LIN {X 0,Y 100.79,Z 485.874,A -85,B 0,C 180,E1 -28454.124,E2 -28454.124} C_VEL
LIN {X 0,Y 100.608,Z 489.017,A -85,B 0,C 180,E1 -28458.321,E2 -28458.321} C_VEL
LIN {X 0,Y 99.957,Z 495.022,A -85,B 0,C 180,E1 -28464.952,E2 -28464.952} C_VEL
LIN {X 0,Y 99.623,Z 497.358,A -85,B 0,C 180,E1 -28467.293,E2 -28467.293} C_VEL
LIN {X 0,Y 98.959,Z 499.354,A -85,B 0,C 180,E1 -28468.917,E2 -28468.917} C_VEL
LIN {X 0,Y 94.552,Z 506.247,A -85,B 0,C 180,E1 -28473.257,E2 -28473.257} C_VEL
LIN {X 0,Y 91.523,Z 510.415,A -85,B 0,C 180,E1 -28476.263,E2 -28476.263} C_VEL
LIN {X 0,Y 84.205,Z 517.353,A -85,B 0,C 180,E1 -28481.307,E2 -28481.307} C_VEL
LIN {X 0,Y 77.66,Z 522.926,A -85,B 0,C 180,E1 -28487.255,E2 -28487.255} C_VEL
LIN {X 0,Y 72.027,Z 527.307,A -85,B 0,C 180,E1 -28494.164,E2 -28494.164} C_VEL
LIN {X 0,Y 68.844,Z 529.631,A -85,B 0,C 180,E1 -28499.307,E2 -28499.307} C_VEL
LIN {X 0,Y 66.338,Z 531.525,A -85,B 0,C 180,E1 -28504.927,E2 -28504.927} C_VEL
LIN {X 0,Y 63.396,Z 533.992,A -85,B 0,C 180,E1 -28517.189,E2 -28517.189} C_VEL
LIN {X 0,Y 62.912,Z 534.633,A -85,B 0,C 180,E1 -28523.585,E2 -28523.585} C_VEL
LIN {X 0,Y 63.099,Z 534.874,A -85,B 0,C 180,E1 -28529.999,E2 -28529.999} C_VEL
LIN {X 0,Y 62.911,Z 534.616,A -85,B 0,C 180,E1 -28536.414,E2 -28536.414} C_VEL
LIN {X 0,Y 63.389,Z 533.964,A -85,B 0,C 180,E1 -28542.811,E2 -28542.811} C_VEL
LIN {X 0,Y 66.335,Z 531.47,A -85,B 0,C 180,E1 -28555.073,E2 -28555.073} C_VEL
LIN {X 0,Y 70.389,Z 528.468,A -85,B 0,C 180,E1 -28563.308,E2 -28563.308} C_VEL
LIN {X 0,Y 75.675,Z 524.426,A -85,B 0,C 180,E1 -28570.549,E2 -28570.549} C_VEL
LIN {X 0,Y 82.981,Z 518.283,A -85,B 0,C 180,E1 -28577.722,E2 -28577.722} C_VEL
LIN {X 0,Y 90.316,Z 511.485,A -85,B 0,C 180,E1 -28582.903,E2 -28582.903} C_VEL
LIN {X 0,Y 93.523,Z 507.46,A -85,B 0,C 180,E1 -28585.753,E2 -28585.753} C_VEL
LIN {X 0,Y 98.232,Z 500.238,A -85,B 0,C 180,E1 -28590.434,E2 -28590.434} C_VEL
LIN {X 0,Y 98.86,Z 499.173,A -85,B 0,C 180,E1 -28591.096,E2 -28591.096} C_VEL
LIN {X 0,Y 99.501,Z 497.198,A -85,B 0,C 180,E1 -28592.701,E2 -28592.701} C_VEL
LIN {X 0,Y 99.98,Z 493.883,A -85,B 0,C 180,E1 -28596.039,E2 -28596.039} C_VEL
LIN {X 0,Y 100.453,Z 488.875,A -85,B 0,C 180,E1 -28601.649,E2 -28601.649} C_VEL
LIN {X 0,Y 100.718,Z 484.543,A -85,B 0,C 180,E1 -28607.663,E2 -28607.663} C_VEL
LIN {X 0,Y 100.776,Z 482.241,A -85,B 0,C 180,E1 -28611.983,E2 -28611.983} C_VEL
LIN {X 0,Y 101.236,Z 479.446,A -85,B 0,C 180,E1 -28620,E2 -28620} C_VEL
LIN {X 0,Y 100.913,Z 479.773,A -85,B 0,C 180,E1 -28623.994,E2 -28623.994} C_VEL
LIN {X 0,Y 100.778,Z 480.51,A -85,B 0,C 180,E1 -28628.018,E2 -28628.018} C_VEL
LIN {X 0,Y 100.794,Z 481.878,A -85,B 0,C 180,E1 -28632.534,E2 -28632.534} C_VEL
LIN {X 0,Y 100.936,Z 484.371,A -85,B 0,C 180,E1 -28638.26,E2 -28638.26} C_VEL
LIN {X 0,Y 101.025,Z 487.017,A -85,B 0,C 180,E1 -28642.783,E2 -28642.783} C_VEL
LIN {X 0,Y 101.064,Z 489.842,A -85,B 0,C 180,E1 -28646.871,E2 -28646.871} C_VEL
LIN {X 0,Y 100.929,Z 493.155,A -85,B 0,C 180,E1 -28651.089,E2 -28651.089} C_VEL
LIN {X 0,Y 100.416,Z 495.894,A -85,B 0,C 180,E1 -28654.05,E2 -28654.05} C_VEL
LIN {X 0,Y 99.593,Z 497.355,A -85,B 0,C 180,E1 -28655.169,E2 -28655.169} C_VEL
LIN {X 0,Y 91.436,Z 505.803,A -85,B 0,C 180,E1 -28659.77,E2 -28659.77} C_VEL
LIN {X 0,Y 84.425,Z 512.165,A -85,B 0,C 180,E1 -28664.961,E2 -28664.961} C_VEL
LIN {X 0,Y 78.061,Z 517.212,A -85,B 0,C 180,E1 -28670.934,E2 -28670.934} C_VEL
LIN {X 0,Y 72.621,Z 521.125,A -85,B 0,C 180,E1 -28677.841,E2 -28677.841} C_VEL
LIN {X 0,Y 68.37,Z 524.004,A -85,B 0,C 180,E1 -28685.722,E2 -28685.722} C_VEL
LIN {X 0,Y 65.957,Z 525.536,A -85,B 0,C 180,E1 -28692.438,E2 -28692.438} C_VEL
LIN {X 0,Y 63.77,Z 526.945,A -85,B 0,C 180,E1 -28703.673,E2 -28703.673} C_VEL
LIN {X 0,Y 63.441,Z 527.168,A -85,B 0,C 180,E1 -28710.001,E2 -28710.001} C_VEL
LIN {X 0,Y 64.129,Z 526.733,A -85,B 0,C 180,E1 -28719.49,E2 -28719.49} C_VEL
LIN {X 0,Y 64.49,Z 526.17,A -85,B 0,C 180,E1 -28724.713,E2 -28724.713} C_VEL
LIN {X 0,Y 64.26,Z 524.809,A -85,B 0,C 180,E1 -28733.474,E2 -28733.474} C_VEL
LIN {X 0,Y 65.296,Z 522.823,A -85,B 0,C 180,E1 -28742.058,E2 -28742.058} C_VEL
LIN {X 0,Y 67.497,Z 521.137,A -85,B 0,C 180,E1 -28746.577,E2 -28746.577} C_VEL
LIN {X 0,Y 74.845,Z 516.238,A -85,B 0,C 180,E1 -28754.771,E2 -28754.771} C_VEL
LIN {X 0,Y 83.182,Z 509.819,A -85,B 0,C 180,E1 -28761.402,E2 -28761.402} C_VEL
LIN {X 0,Y 91.092,Z 502.744,A -85,B 0,C 180,E1 -28766.038,E2 -28766.038} C_VEL
LIN {X 0,Y 94.19,Z 499.661,A -85,B 0,C 180,E1 -28767.608,E2 -28767.608} C_VEL
LIN {X 0,Y 95.055,Z 498.216,A -85,B 0,C 180,E1 -28768.831,E2 -28768.831} C_VEL
LIN {X 0,Y 95.682,Z 494.585,A -85,B 0,C 180,E1 -28773.85,E2 -28773.85} C_VEL
LIN {X 0,Y 96.006,Z 491.648,A -85,B 0,C 180,E1 -28778.529,E2 -28778.529} C_VEL
LIN {X 0,Y 96.173,Z 489.36,A -85,B 0,C 180,E1 -28783.004,E2 -28783.004} C_VEL
LIN {X 0,Y 96.285,Z 487.591,A -85,B 0,C 180,E1 -28787.351,E2 -28787.351} C_VEL
LIN {X 0,Y 96.396,Z 486.427,A -85,B 0,C 180,E1 -28791.615,E2 -28791.615} C_VEL
LIN {X 0,Y 96.593,Z 485.676,A -85,B 0,C 180,E1 -28795.827,E2 -28795.827} C_VEL
LIN {X 0,Y 96.879,Z 485.44,A -85,B 0,C 180,E1 -28800,E2 -28800} C_VEL
LIN {X 0,Y 96.468,Z 486.677,A -85,B 0,C 180,E1 -28804.178,E2 -28804.178} C_VEL
LIN {X 0,Y 96.276,Z 488.267,A -85,B 0,C 180,E1 -28808.395,E2 -28808.395} C_VEL
LIN {X 0,Y 95.961,Z 490.508,A -85,B 0,C 180,E1 -28812.692,E2 -28812.692} C_VEL
LIN {X 0,Y 95.505,Z 493.514,A -85,B 0,C 180,E1 -28817.119,E2 -28817.119} C_VEL
LIN {X 0,Y 94.742,Z 497.275,A -85,B 0,C 180,E1 -28821.771,E2 -28821.771} C_VEL
LIN {X 0,Y 93.803,Z 501.058,A -85,B 0,C 180,E1 -28825.961,E2 -28825.961} C_VEL
LIN {X 0,Y 92.38,Z 503.337,A -85,B 0,C 180,E1 -28827.603,E2 -28827.603} C_VEL
LIN {X 0,Y 86.175,Z 511.231,A -85,B 0,C 180,E1 -28833.285,E2 -28833.285} C_VEL
LIN {X 0,Y 78.294,Z 518.042,A -85,B 0,C 180,E1 -28838.445,E2 -28838.445} C_VEL
LIN {X 0,Y 70.403,Z 524.098,A -85,B 0,C 180,E1 -28845.67,E2 -28845.67} C_VEL
LIN {X 0,Y 64.534,Z 528.111,A -85,B 0,C 180,E1 -28853.203,E2 -28853.203} C_VEL
LIN {X 0,Y 59.936,Z 531.09,A -85,B 0,C 180,E1 -28862.028,E2 -28862.028} C_VEL
LIN {X 0,Y 56.464,Z 533.558,A -85,B 0,C 180,E1 -28875.584,E2 -28875.584} C_VEL
LIN {X 0,Y 55.837,Z 534.199,A -85,B 0,C 180,E1 -28882.768,E2 -28882.768} C_VEL
LIN {X 0,Y 56.013,Z 534.443,A -85,B 0,C 180,E1 -28889.999,E2 -28889.999} C_VEL
LIN {X 0,Y 55.836,Z 534.182,A -85,B 0,C 180,E1 -28897.23,E2 -28897.23} C_VEL
LIN {X 0,Y 56.456,Z 533.53,A -85,B 0,C 180,E1 -28904.416,E2 -28904.416} C_VEL
LIN {X 0,Y 57.815,Z 532.484,A -85,B 0,C 180,E1 -28911.387,E2 -28911.387} C_VEL
LIN {X 0,Y 59.933,Z 531.034,A -85,B 0,C 180,E1 -28917.972,E2 -28917.972} C_VEL
LIN {X 0,Y 64.532,Z 528.031,A -85,B 0,C 180,E1 -28926.797,E2 -28926.797} C_VEL
LIN {X 0,Y 70.405,Z 523.99,A -85,B 0,C 180,E1 -28934.327,E2 -28934.327} C_VEL
LIN {X 0,Y 78.294,Z 517.891,A -85,B 0,C 180,E1 -28941.553,E2 -28941.553} C_VEL
LIN {X 0,Y 86.139,Z 511.041,A -85,B 0,C 180,E1 -28946.749,E2 -28946.749} C_VEL
LIN {X 0,Y 91.267,Z 504.579,A -85,B 0,C 180,E1 -28951.468,E2 -28951.468} C_VEL
LIN {X 0,Y 92.954,Z 502.244,A -85,B 0,C 180,E1 -28953.022,E2 -28953.022} C_VEL
LIN {X 0,Y 93.735,Z 500.797,A -85,B 0,C 180,E1 -28954.122,E2 -28954.122} C_VEL
LIN {X 0,Y 94.286,Z 498.915,A -85,B 0,C 180,E1 -28956.085,E2 -28956.085} C_VEL
LIN {X 0,Y 95.413,Z 493.079,A -85,B 0,C 180,E1 -28963.248,E2 -28963.248} C_VEL
LIN {X 0,Y 95.862,Z 490.299,A -85,B 0,C 180,E1 -28967.295,E2 -28967.295} C_VEL
LIN {X 0,Y 96.188,Z 488.023,A -85,B 0,C 180,E1 -28971.597,E2 -28971.597} C_VEL
LIN {X 0,Y 96.8,Z 485.161,A -85,B 0,C 180,E1 -28980,E2 -28980} C_VEL
LIN {X 0,Y 96.484,Z 485.426,A -85,B 0,C 180,E1 -28984.177,E2 -28984.177} C_VEL
LIN {X 0,Y 96.277,Z 486.19,A -85,B 0,C 180,E1 -28988.395,E2 -28988.395} C_VEL
LIN {X 0,Y 96.129,Z 487.408,A -85,B 0,C 180,E1 -28992.67,E2 -28992.67} C_VEL
LIN {X 0,Y 96.043,Z 489.575,A -85,B 0,C 180,E1 -28997.958,E2 -28997.958} C_VEL
LIN {X 0,Y 95.855,Z 492.741,A -85,B 0,C 180,E1 -29003.782,E2 -29003.782} C_VEL
LIN {X 0,Y 95.322,Z 496.692,A -85,B 0,C 180,E1 -29009.528,E2 -29009.528} C_VEL
LIN {X 0,Y 95.04,Z 497.937,A -85,B 0,C 180,E1 -29011.174,E2 -29011.174} C_VEL
LIN {X 0,Y 94.182,Z 499.388,A -85,B 0,C 180,E1 -29012.417,E2 -29012.417} C_VEL
LIN {X 0,Y 87.085,Z 506.235,A -85,B 0,C 180,E1 -29016.194,E2 -29016.194} C_VEL
LIN {X 0,Y 79.563,Z 512.6,A -85,B 0,C 180,E1 -29021.338,E2 -29021.338} C_VEL
LIN {X 0,Y 72.695,Z 517.645,A -85,B 0,C 180,E1 -29027.41,E2 -29027.41} C_VEL
LIN {X 0,Y 66.725,Z 521.558,A -85,B 0,C 180,E1 -29034.599,E2 -29034.599} C_VEL
LIN {X 0,Y 61.993,Z 524.435,A -85,B 0,C 180,E1 -29043.034,E2 -29043.034} C_VEL
LIN {X 0,Y 57.871,Z 526.776,A -85,B 0,C 180,E1 -29055.944,E2 -29055.944} C_VEL
LIN {X 0,Y 56.355,Z 527.599,A -85,B 0,C 180,E1 -29070.001,E2 -29070.001} C_VEL
LIN {X 0,Y 57.133,Z 527.138,A -85,B 0,C 180,E1 -29080.505,E2 -29080.505} C_VEL
LIN {X 0,Y 59.525,Z 525.861,A -85,B 0,C 180,E1 -29090.745,E2 -29090.745} C_VEL
LIN {X 0,Y 61.929,Z 524.516,A -85,B 0,C 180,E1 -29096.998,E2 -29096.998} C_VEL
LIN {X 0,Y 67.497,Z 521.137,A -85,B 0,C 180,E1 -29106.577,E2 -29106.577} C_VEL
LIN {X 0,Y 70.032,Z 519.236,A -85,B 0,C 180,E1 -29110.727,E2 -29110.727} C_VEL
LIN {X 0,Y 74.825,Z 514.222,A -85,B 0,C 180,E1 -29120.276,E2 -29120.276} C_VEL
LIN {X 0,Y 78.484,Z 510.721,A -85,B 0,C 180,E1 -29124.827,E2 -29124.827} C_VEL
LIN {X 0,Y 80.858,Z 508.702,A -85,B 0,C 180,E1 -29126.573,E2 -29126.573} C_VEL
LIN {X 0,Y 88.77,Z 501.83,A -85,B 0,C 180,E1 -29130.562,E2 -29130.562} C_VEL
LIN {X 0,Y 89.663,Z 500.503,A -85,B 0,C 180,E1 -29131.946,E2 -29131.946} C_VEL
LIN {X 0,Y 90.487,Z 497.322,A -85,B 0,C 180,E1 -29137.148,E2 -29137.148} C_VEL
LIN {X 0,Y 90.879,Z 494.942,A -85,B 0,C 180,E1 -29141.981,E2 -29141.981} C_VEL
LIN {X 0,Y 91.222,Z 493.097,A -85,B 0,C 180,E1 -29146.636,E2 -29146.636} C_VEL
LIN {X 0,Y 91.515,Z 491.822,A -85,B 0,C 180,E1 -29151.165,E2 -29151.165} C_VEL
LIN {X 0,Y 91.848,Z 491.066,A -85,B 0,C 180,E1 -29155.611,E2 -29155.611} C_VEL
LIN {X 0,Y 92.125,Z 490.89,A -85,B 0,C 180,E1 -29160,E2 -29160} C_VEL
LIN {X 0,Y 91.618,Z 492.162,A -85,B 0,C 180,E1 -29164.399,E2 -29164.399} C_VEL
LIN {X 0,Y 91.239,Z 493.806,A -85,B 0,C 180,E1 -29168.862,E2 -29168.862} C_VEL
LIN {X 0,Y 90.59,Z 496.306,A -85,B 0,C 180,E1 -29173.458,E2 -29173.458} C_VEL
LIN {X 0,Y 89.658,Z 499.533,A -85,B 0,C 180,E1 -29178.273,E2 -29178.273} C_VEL
LIN {X 0,Y 88.326,Z 503.575,A -85,B 0,C 180,E1 -29183.443,E2 -29183.443} C_VEL
LIN {X 0,Y 85.891,Z 506.74,A -85,B 0,C 180,E1 -29185.831,E2 -29185.831} C_VEL
LIN {X 0,Y 81.064,Z 512.044,A -85,B 0,C 180,E1 -29189.89,E2 -29189.89} C_VEL
LIN {X 0,Y 72.884,Z 518.508,A -85,B 0,C 180,E1 -29194.95,E2 -29194.95} C_VEL
LIN {X 0,Y 65.483,Z 523.664,A -85,B 0,C 180,E1 -29201.297,E2 -29201.297} C_VEL
LIN {X 0,Y 58.968,Z 527.676,A -85,B 0,C 180,E1 -29209.041,E2 -29209.041} C_VEL
LIN {X 0,Y 53.727,Z 530.655,A -85,B 0,C 180,E1 -29218.449,E2 -29218.449} C_VEL
LIN {X 0,Y 51.245,Z 532.089,A -85,B 0,C 180,E1 -29225.704,E2 -29225.704} C_VEL
LIN {X 0,Y 48.798,Z 533.767,A -85,B 0,C 180,E1 -29241.718,E2 -29241.718} C_VEL
LIN {X 0,Y 48.912,Z 534.01,A -85,B 0,C 180,E1 -29249.999,E2 -29249.999} C_VEL
LIN {X 0,Y 48.796,Z 533.749,A -85,B 0,C 180,E1 -29258.28,E2 -29258.28} C_VEL
LIN {X 0,Y 51.235,Z 532.049,A -85,B 0,C 180,E1 -29274.299,E2 -29274.299} C_VEL
LIN {X 0,Y 53.725,Z 530.598,A -85,B 0,C 180,E1 -29281.55,E2 -29281.55} C_VEL
LIN {X 0,Y 58.966,Z 527.595,A -85,B 0,C 180,E1 -29290.959,E2 -29290.959} C_VEL
LIN {X 0,Y 65.487,Z 523.554,A -85,B 0,C 180,E1 -29298.697,E2 -29298.697} C_VEL
LIN {X 0,Y 74.066,Z 517.454,A -85,B 0,C 180,E1 -29305.883,E2 -29305.883} C_VEL
LIN {X 0,Y 81.05,Z 511.853,A -85,B 0,C 180,E1 -29310.125,E2 -29310.125} C_VEL
LIN {X 0,Y 85.842,Z 506.522,A -85,B 0,C 180,E1 -29314.234,E2 -29314.234} C_VEL
LIN {X 0,Y 88.241,Z 503.419,A -85,B 0,C 180,E1 -29316.533,E2 -29316.533} C_VEL
LIN {X 0,Y 89.321,Z 500.093,A -85,B 0,C 180,E1 -29320.768,E2 -29320.768} C_VEL
LIN {X 0,Y 90.506,Z 496.101,A -85,B 0,C 180,E1 -29326.529,E2 -29326.529} C_VEL
LIN {X 0,Y 91.149,Z 493.599,A -85,B 0,C 180,E1 -29331.129,E2 -29331.129} C_VEL
LIN {X 0,Y 91.589,Z 491.785,A -85,B 0,C 180,E1 -29335.983,E2 -29335.983} C_VEL
LIN {X 0,Y 92.057,Z 490.624,A -85,B 0,C 180,E1 -29340,E2 -29340} C_VEL
LIN {X 0,Y 91.693,Z 490.915,A -85,B 0,C 180,E1 -29344.858,E2 -29344.858} C_VEL
LIN {X 0,Y 91.395,Z 491.623,A -85,B 0,C 180,E1 -29348.847,E2 -29348.847} C_VEL
LIN {X 0,Y 91.091,Z 492.905,A -85,B 0,C 180,E1 -29353.383,E2 -29353.383} C_VEL
LIN {X 0,Y 90.797,Z 494.716,A -85,B 0,C 180,E1 -29358.036,E2 -29358.036} C_VEL
LIN {X 0,Y 90.415,Z 497.089,A -85,B 0,C 180,E1 -29362.871,E2 -29362.871} C_VEL
LIN {X 0,Y 89.632,Z 500.246,A -85,B 0,C 180,E1 -29368.064,E2 -29368.064} C_VEL
LIN {X 0,Y 88.767,Z 501.567,A -85,B 0,C 180,E1 -29369.436,E2 -29369.436} C_VEL
LIN {X 0,Y 80.356,Z 508.93,A -85,B 0,C 180,E1 -29373.811,E2 -29373.811} C_VEL
LIN {X 0,Y 72.527,Z 514.826,A -85,B 0,C 180,E1 -29379.176,E2 -29379.176} C_VEL
LIN {X 0,Y 65.341,Z 519.485,A -85,B 0,C 180,E1 -29385.643,E2 -29385.643} C_VEL
LIN {X 0,Y 59.166,Z 523.039,A -85,B 0,C 180,E1 -29393.564,E2 -29393.564} C_VEL
LIN {X 0,Y 55.759,Z 524.868,A -85,B 0,C 180,E1 -29399.724,E2 -29399.724} C_VEL
LIN {X 0,Y 51.022,Z 527.208,A -85,B 0,C 180,E1 -29414.01,E2 -29414.01} C_VEL
LIN {X 0,Y 49.735,Z 527.807,A -85,B 0,C 180,E1 -29421.877,E2 -29421.877} C_VEL
LIN {X 0,Y 49.285,Z 528.03,A -85,B 0,C 180,E1 -29430.001,E2 -29430.001} C_VEL
LIN {X 0,Y 49.696,Z 527.833,A -85,B 0,C 180,E1 -29438.131,E2 -29438.131} C_VEL
LIN {X 0,Y 50.97,Z 527.249,A -85,B 0,C 180,E1 -29446.009,E2 -29446.009} C_VEL
LIN {X 0,Y 55.697,Z 524.948,A -85,B 0,C 180,E1 -29460.315,E2 -29460.315} C_VEL
LIN {X 0,Y 61.724,Z 521.703,A -85,B 0,C 180,E1 -29470.176,E2 -29470.176} C_VEL
LIN {X 0,Y 67.598,Z 518.224,A -85,B 0,C 180,E1 -29476.701,E2 -29476.701} C_VEL
LIN {X 0,Y 75.001,Z 513.223,A -85,B 0,C 180,E1 -29482.798,E2 -29482.798} C_VEL
LIN {X 0,Y 80.858,Z 508.702,A -85,B 0,C 180,E1 -29486.573,E2 -29486.573} C_VEL
LIN {X 0,Y 82.872,Z 506.727,A -85,B 0,C 180,E1 -29488.471,E2 -29488.471} C_VEL
LIN {X 0,Y 84,Z 504.998,A -85,B 0,C 180,E1 -29490.825,E2 -29490.825} C_VEL
LIN {X 0,Y 84.635,Z 503.095,A -85,B 0,C 180,E1 -29494.337,E2 -29494.337} C_VEL
LIN {X 0,Y 85.088,Z 500.631,A -85,B 0,C 180,E1 -29499.899,E2 -29499.899} C_VEL
LIN {X 0,Y 85.78,Z 498.382,A -85,B 0,C 180,E1 -29505.771,E2 -29505.771} C_VEL
LIN {X 0,Y 86.279,Z 496.992,A -85,B 0,C 180,E1 -29510.624,E2 -29510.624} C_VEL
LIN {X 0,Y 86.78,Z 496.15,A -85,B 0,C 180,E1 -29515.354,E2 -29515.354} C_VEL
LIN {X 0,Y 87.049,Z 496.062,A -85,B 0,C 180,E1 -29520,E2 -29520} C_VEL
LIN {X 0,Y 86.402,Z 497.351,A -85,B 0,C 180,E1 -29524.665,E2 -29524.665} C_VEL
LIN {X 0,Y 85.676,Z 499.486,A -85,B 0,C 180,E1 -29530.141,E2 -29530.141} C_VEL
LIN {X 0,Y 84.743,Z 501.842,A -85,B 0,C 180,E1 -29534.406,E2 -29534.406} C_VEL
LIN {X 0,Y 83.267,Z 505.353,A -85,B 0,C 180,E1 -29539.731,E2 -29539.731} C_VEL
LIN {X 0,Y 82.782,Z 506.266,A -85,B 0,C 180,E1 -29540.951,E2 -29540.951} C_VEL
LIN {X 0,Y 77.619,Z 511.592,A -85,B 0,C 180,E1 -29545.115,E2 -29545.115} C_VEL
LIN {X 0,Y 74.804,Z 513.903,A -85,B 0,C 180,E1 -29546.803,E2 -29546.803} C_VEL
LIN {X 0,Y 65.546,Z 520.376,A -85,B 0,C 180,E1 -29552.419,E2 -29552.419} C_VEL
LIN {X 0,Y 58.469,Z 524.679,A -85,B 0,C 180,E1 -29558.619,E2 -29558.619} C_VEL
LIN {X 0,Y 51.638,Z 528.333,A -85,B 0,C 180,E1 -29567.116,E2 -29567.116} C_VEL
LIN {X 0,Y 47.785,Z 530.221,A -85,B 0,C 180,E1 -29573.962,E2 -29573.962} C_VEL
LIN {X 0,Y 42.791,Z 532.69,A -85,B 0,C 180,E1 -29590.822,E2 -29590.822} C_VEL
LIN {X 0,Y 41.755,Z 533.333,A -85,B 0,C 180,E1 -29600.309,E2 -29600.309} C_VEL
LIN {X 0,Y 41.821,Z 533.578,A -85,B 0,C 180,E1 -29609.999,E2 -29609.999} C_VEL
LIN {X 0,Y 42.785,Z 532.66,A -85,B 0,C 180,E1 -29629.179,E2 -29629.179} C_VEL
LIN {X 0,Y 47.782,Z 530.162,A -85,B 0,C 180,E1 -29646.038,E2 -29646.038} C_VEL
LIN {X 0,Y 53.776,Z 527.159,A -85,B 0,C 180,E1 -29655.955,E2 -29655.955} C_VEL
LIN {X 0,Y 62.658,Z 522.062,A -85,B 0,C 180,E1 -29665.264,E2 -29665.264} C_VEL
LIN {X 0,Y 71.875,Z 515.894,A -85,B 0,C 180,E1 -29671.645,E2 -29671.645} C_VEL
LIN {X 0,Y 76.262,Z 512.597,A -85,B 0,C 180,E1 -29673.963,E2 -29673.963} C_VEL
LIN {X 0,Y 81.464,Z 507.457,A -85,B 0,C 180,E1 -29678.036,E2 -29678.036} C_VEL
LIN {X 0,Y 82.749,Z 506.045,A -85,B 0,C 180,E1 -29679.106,E2 -29679.106} C_VEL
LIN {X 0,Y 83.909,Z 503.381,A -85,B 0,C 180,E1 -29682.954,E2 -29682.954} C_VEL
LIN {X 0,Y 85.307,Z 500.071,A -85,B 0,C 180,E1 -29688.355,E2 -29688.355} C_VEL
LIN {X 0,Y 85.744,Z 498.922,A -85,B 0,C 180,E1 -29690.565,E2 -29690.565} C_VEL
LIN {X 0,Y 86.342,Z 497.128,A -85,B 0,C 180,E1 -29695.331,E2 -29695.331} C_VEL
LIN {X 0,Y 87.016,Z 495.805,A -85,B 0,C 180,E1 -29700,E2 -29700} C_VEL
LIN {X 0,Y 86.677,Z 495.956,A -85,B 0,C 180,E1 -29704.651,E2 -29704.651} C_VEL
LIN {X 0,Y 85.99,Z 497.261,A -85,B 0,C 180,E1 -29711.255,E2 -29711.255} C_VEL
LIN {X 0,Y 85.688,Z 498.179,A -85,B 0,C 180,E1 -29714.244,E2 -29714.244} C_VEL
LIN {X 0,Y 84.919,Z 500.872,A -85,B 0,C 180,E1 -29721.174,E2 -29721.174} C_VEL
LIN {X 0,Y 84.273,Z 502.635,A -85,B 0,C 180,E1 -29724.644,E2 -29724.644} C_VEL
LIN {X 0,Y 83.455,Z 503.85,A -85,B 0,C 180,E1 -29726.195,E2 -29726.195} C_VEL
LIN {X 0,Y 73.763,Z 511.486,A -85,B 0,C 180,E1 -29730.963,E2 -29730.963} C_VEL
LIN {X 0,Y 65.588,Z 516.938,A -85,B 0,C 180,E1 -29736.521,E2 -29736.521} C_VEL
LIN {X 0,Y 58.077,Z 521.214,A -85,B 0,C 180,E1 -29743.443,E2 -29743.443} C_VEL
LIN {X 0,Y 53.63,Z 523.471,A -85,B 0,C 180,E1 -29749.063,E2 -29749.063} C_VEL
LIN {X 0,Y 49.757,Z 525.301,A -85,B 0,C 180,E1 -29755.599,E2 -29755.599} C_VEL
LIN {X 0,Y 46.604,Z 526.668,A -85,B 0,C 180,E1 -29763.103,E2 -29763.103} C_VEL
LIN {X 0,Y 44.257,Z 527.64,A -85,B 0,C 180,E1 -29771.483,E2 -29771.483} C_VEL
LIN {X 0,Y 42.75,Z 528.238,A -85,B 0,C 180,E1 -29780.539,E2 -29780.539} C_VEL
LIN {X 0,Y 42.314,Z 528.394,A -85,B 0,C 180,E1 -29794.76,E2 -29794.76} C_VEL
LIN {X 0,Y 44.207,Z 527.68,A -85,B 0,C 180,E1 -29808.541,E2 -29808.541} C_VEL
LIN {X 0,Y 49.708,Z 525.379,A -85,B 0,C 180,E1 -29824.442,E2 -29824.442} C_VEL
LIN {X 0,Y 55.75,Z 522.529,A -85,B 0,C 180,E1 -29833.897,E2 -29833.897} C_VEL
LIN {X 0,Y 62.943,Z 518.655,A -85,B 0,C 180,E1 -29841.409,E2 -29841.409} C_VEL
LIN {X 0,Y 70.941,Z 513.653,A -85,B 0,C 180,E1 -29847.362,E2 -29847.362} C_VEL
LIN {X 0,Y 79.519,Z 507.341,A -85,B 0,C 180,E1 -29852.108,E2 -29852.108} C_VEL
LIN {X 0,Y 83.459,Z 504.092,A -85,B 0,C 180,E1 -29853.84,E2 -29853.84} C_VEL
LIN {X 0,Y 84.281,Z 502.887,A -85,B 0,C 180,E1 -29855.358,E2 -29855.358} C_VEL
LIN {X 0,Y 85.088,Z 500.631,A -85,B 0,C 180,E1 -29859.899,E2 -29859.899} C_VEL
LIN {X 0,Y 84.837,Z 500.012,A -85,B 0,C 180,E1 -29862.492,E2 -29862.492} C_VEL
LIN {X 0,Y 83.477,Z 500.26,A -85,B 0,C 180,E1 -29865.992,E2 -29865.992} C_VEL
LIN {X 0,Y 81.365,Z 501.197,A -85,B 0,C 180,E1 -29871.491,E2 -29871.491} C_VEL
LIN {X 0,Y 81.271,Z 501.097,A -85,B 0,C 180,E1 -29874.366,E2 -29874.366} C_VEL
LIN {X 0,Y 81.659,Z 500.92,A -85,B 0,C 180,E1 -29880,E2 -29880} C_VEL
LIN {X 0,Y 80.854,Z 502.285,A -85,B 0,C 180,E1 -29884.986,E2 -29884.986} C_VEL
LIN {X 0,Y 79.936,Z 504.259,A -85,B 0,C 180,E1 -29890.127,E2 -29890.127} C_VEL
LIN {X 0,Y 78.277,Z 507.234,A -85,B 0,C 180,E1 -29895.626,E2 -29895.626} C_VEL
LIN {X 0,Y 77.328,Z 508.734,A -85,B 0,C 180,E1 -29897.933,E2 -29897.933} C_VEL
LIN {X 0,Y 73.322,Z 512.324,A -85,B 0,C 180,E1 -29900.843,E2 -29900.843} C_VEL
LIN {X 0,Y 68.774,Z 515.618,A -85,B 0,C 180,E1 -29903.114,E2 -29903.114} C_VEL
LIN {X 0,Y 59.806,Z 521.205,A -85,B 0,C 180,E1 -29908.286,E2 -29908.286} C_VEL
LIN {X 0,Y 51.619,Z 525.568,A -85,B 0,C 180,E1 -29915.221,E2 -29915.221} C_VEL
LIN {X 0,Y 46.653,Z 527.898,A -85,B 0,C 180,E1 -29921.128,E2 -29921.128} C_VEL
LIN {X 0,Y 42.219,Z 529.787,A -85,B 0,C 180,E1 -29928.25,E2 -29928.25} C_VEL
LIN {X 0,Y 36.143,Z 532.256,A -85,B 0,C 180,E1 -29947.113,E2 -29947.113} C_VEL
LIN {X 0,Y 34.717,Z 533.146,A -85,B 0,C 180,E1 -29969.999,E2 -29969.999} C_VEL
LIN {X 0,Y 36.111,Z 532.225,A -85,B 0,C 180,E1 -29992.906,E2 -29992.906} C_VEL
LIN {X 0,Y 42.217,Z 529.727,A -85,B 0,C 180,E1 -30011.75,E2 -30011.75} C_VEL
LIN {X 0,Y 49.08,Z 526.724,A -85,B 0,C 180,E1 -30021.958,E2 -30021.958} C_VEL
LIN {X 0,Y 57.049,Z 522.678,A -85,B 0,C 180,E1 -30029.581,E2 -30029.581} C_VEL
LIN {X 0,Y 65.751,Z 517.491,A -85,B 0,C 180,E1 -30035.306,E2 -30035.306} C_VEL
LIN {X 0,Y 71.86,Z 513.29,A -85,B 0,C 180,E1 -30038.296,E2 -30038.296} C_VEL
LIN {X 0,Y 77.268,Z 508.561,A -85,B 0,C 180,E1 -30042.097,E2 -30042.097} C_VEL
LIN {X 0,Y 78.148,Z 507.114,A -85,B 0,C 180,E1 -30044.348,E2 -30044.348} C_VEL
LIN {X 0,Y 79.863,Z 504.084,A -85,B 0,C 180,E1 -30049.863,E2 -30049.863} C_VEL
LIN {X 0,Y 80.786,Z 502.088,A -85,B 0,C 180,E1 -30055.009,E2 -30055.009} C_VEL
LIN {X 0,Y 81.624,Z 500.69,A -85,B 0,C 180,E1 -30060,E2 -30060} C_VEL
LIN {X 0,Y 81.284,Z 500.804,A -85,B 0,C 180,E1 -30064.96,E2 -30064.96} C_VEL
LIN {X 0,Y 80.689,Z 501.663,A -85,B 0,C 180,E1 -30070.032,E2 -30070.032} C_VEL
LIN {X 0,Y 79.878,Z 503.149,A -85,B 0,C 180,E1 -30075.305,E2 -30075.305} C_VEL
LIN {X 0,Y 79.04,Z 505.144,A -85,B 0,C 180,E1 -30080.835,E2 -30080.835} C_VEL
LIN {X 0,Y 78.218,Z 506.186,A -85,B 0,C 180,E1 -30082.588,E2 -30082.588} C_VEL
LIN {X 0,Y 70.379,Z 511.92,A -85,B 0,C 180,E1 -30086.008,E2 -30086.008} C_VEL
LIN {X 0,Y 61.634,Z 517.371,A -85,B 0,C 180,E1 -30091.218,E2 -30091.218} C_VEL
LIN {X 0,Y 53.46,Z 521.646,A -85,B 0,C 180,E1 -30097.929,E2 -30097.929} C_VEL
LIN {X 0,Y 48.505,Z 523.903,A -85,B 0,C 180,E1 -30103.577,E2 -30103.577} C_VEL
LIN {X 0,Y 44.091,Z 525.733,A -85,B 0,C 180,E1 -30110.388,E2 -30110.388} C_VEL
LIN {X 0,Y 40.411,Z 527.101,A -85,B 0,C 180,E1 -30118.552,E2 -30118.552} C_VEL
LIN {X 0,Y 37.609,Z 528.071,A -85,B 0,C 180,E1 -30128.055,E2 -30128.055} C_VEL
LIN {X 0,Y 35.799,Z 528.668,A -85,B 0,C 180,E1 -30138.68,E2 -30138.68} C_VEL
LIN {X 0,Y 35.14,Z 528.891,A -85,B 0,C 180,E1 -30150.001,E2 -30150.001} C_VEL
LIN {X 0,Y 35.754,Z 528.693,A -85,B 0,C 180,E1 -30161.338,E2 -30161.338} C_VEL
LIN {X 0,Y 37.549,Z 528.111,A -85,B 0,C 180,E1 -30171.985,E2 -30171.985} C_VEL
LIN {X 0,Y 44.054,Z 525.809,A -85,B 0,C 180,E1 -30189.653,E2 -30189.653} C_VEL
LIN {X 0,Y 50.877,Z 522.96,A -85,B 0,C 180,E1 -30199.444,E2 -30199.444} C_VEL
LIN {X 0,Y 58.781,Z 519.086,A -85,B 0,C 180,E1 -30206.82,E2 -30206.82} C_VEL
LIN {X 0,Y 67.385,Z 514.083,A -85,B 0,C 180,E1 -30212.44,E2 -30212.44} C_VEL
LIN {X 0,Y 76.467,Z 507.769,A -85,B 0,C 180,E1 -30216.796,E2 -30216.796} C_VEL
LIN {X 0,Y 78.26,Z 506.379,A -85,B 0,C 180,E1 -30217.45,E2 -30217.45} C_VEL
LIN {X 0,Y 79.047,Z 505.371,A -85,B 0,C 180,E1 -30219.167,E2 -30219.167} C_VEL
LIN {X 0,Y 79.588,Z 504.23,A -85,B 0,C 180,E1 -30221.997,E2 -30221.997} C_VEL
LIN {X 0,Y 80.786,Z 501.849,A -85,B 0,C 180,E1 -30229.98,E2 -30229.98} C_VEL
LIN {X 0,Y 81.271,Z 501.097,A -85,B 0,C 180,E1 -30234.366,E2 -30234.366} C_VEL
LIN {X 0,Y 81.137,Z 501.199,A -85,B 0,C 180,E1 -30236.608,E2 -30236.608} C_VEL
LIN {X 0,Y 79.834,Z 502.442,A -85,B 0,C 180,E1 -30239.604,E2 -30239.604} C_VEL
LIN {X 0,Y 74.297,Z 507.987,A -85,B 0,C 180,E1 -30248.344,E2 -30248.344} C_VEL
LIN {X 0,Y 73.466,Z 509.167,A -85,B 0,C 180,E1 -30251.03,E2 -30251.03} C_VEL
LIN {X 0,Y 72.392,Z 510.647,A -85,B 0,C 180,E1 -30253.871,E2 -30253.871} C_VEL
LIN {X 0,Y 69.48,Z 513.023,A -85,B 0,C 180,E1 -30256.063,E2 -30256.063} C_VEL
LIN {X 0,Y 63.103,Z 517.208,A -85,B 0,C 180,E1 -30258.793,E2 -30258.793} C_VEL
LIN {X 0,Y 53.766,Z 522.357,A -85,B 0,C 180,E1 -30263.792,E2 -30263.792} C_VEL
LIN {X 0,Y 45.035,Z 526.374,A -85,B 0,C 180,E1 -30270.871,E2 -30270.871} C_VEL
LIN {X 0,Y 37.195,Z 529.352,A -85,B 0,C 180,E1 -30280.903,E2 -30280.903} C_VEL
LIN {X 0,Y 29.692,Z 531.822,A -85,B 0,C 180,E1 -30301.744,E2 -30301.744} C_VEL
LIN {X 0,Y 27.834,Z 532.467,A -85,B 0,C 180,E1 -30315.373,E2 -30315.373} C_VEL
LIN {X 0,Y 27.596,Z 532.712,A -85,B 0,C 180,E1 -30329.999,E2 -30329.999} C_VEL
LIN {X 0,Y 27.829,Z 532.448,A -85,B 0,C 180,E1 -30344.626,E2 -30344.626} C_VEL
LIN {X 0,Y 32.906,Z 530.743,A -85,B 0,C 180,E1 -30369.845,E2 -30369.845} C_VEL
LIN {X 0,Y 37.193,Z 529.291,A -85,B 0,C 180,E1 -30379.098,E2 -30379.098} C_VEL
LIN {X 0,Y 45.034,Z 526.288,A -85,B 0,C 180,E1 -30389.129,E2 -30389.129} C_VEL
LIN {X 0,Y 53.771,Z 522.24,A -85,B 0,C 180,E1 -30396.193,E2 -30396.193} C_VEL
LIN {X 0,Y 64.688,Z 516.041,A -85,B 0,C 180,E1 -30401.922,E2 -30401.922} C_VEL
LIN {X 0,Y 69.469,Z 512.839,A -85,B 0,C 180,E1 -30403.965,E2 -30403.965} C_VEL
LIN {X 0,Y 70.962,Z 511.678,A -85,B 0,C 180,E1 -30404.933,E2 -30404.933} C_VEL
LIN {X 0,Y 72.347,Z 510.433,A -85,B 0,C 180,E1 -30406.27,E2 -30406.27} C_VEL
LIN {X 0,Y 74.313,Z 507.728,A -85,B 0,C 180,E1 -30411.845,E2 -30411.845} C_VEL
LIN {X 0,Y 75.935,Z 505.296,A -85,B 0,C 180,E1 -30420,E2 -30420} C_VEL
LIN {X 0,Y 75.614,Z 505.365,A -85,B 0,C 180,E1 -30425.333,E2 -30425.333} C_VEL
LIN {X 0,Y 74.762,Z 506.316,A -85,B 0,C 180,E1 -30430.837,E2 -30430.837} C_VEL
LIN {X 0,Y 73.548,Z 508.056,A -85,B 0,C 180,E1 -30437.144,E2 -30437.144} C_VEL
LIN {X 0,Y 72.813,Z 508.82,A -85,B 0,C 180,E1 -30438.605,E2 -30438.605} C_VEL
LIN {X 0,Y 64.447,Z 514.334,A -85,B 0,C 180,E1 -30442.04,E2 -30442.04} C_VEL
LIN {X 0,Y 55.253,Z 519.378,A -85,B 0,C 180,E1 -30447.081,E2 -30447.081} C_VEL
LIN {X 0,Y 46.613,Z 523.288,A -85,B 0,C 180,E1 -30453.98,E2 -30453.98} C_VEL
LIN {X 0,Y 38.902,Z 526.165,A -85,B 0,C 180,E1 -30463.729,E2 -30463.729} C_VEL
LIN {X 0,Y 31.143,Z 528.503,A -85,B 0,C 180,E1 -30483.171,E2 -30483.171} C_VEL
LIN {X 0,Y 28.895,Z 529.099,A -85,B 0,C 180,E1 -30495.925,E2 -30495.925} C_VEL
LIN {X 0,Y 28.075,Z 529.322,A -85,B 0,C 180,E1 -30510.001,E2 -30510.001} C_VEL
LIN {X 0,Y 28.838,Z 529.125,A -85,B 0,C 180,E1 -30524.107,E2 -30524.107} C_VEL
LIN {X 0,Y 31.094,Z 528.542,A -85,B 0,C 180,E1 -30536.877,E2 -30536.877} C_VEL
LIN {X 0,Y 38.858,Z 526.24,A -85,B 0,C 180,E1 -30556.342,E2 -30556.342} C_VEL
LIN {X 0,Y 46.583,Z 523.39,A -85,B 0,C 180,E1 -30566.08,E2 -30566.08} C_VEL
LIN {X 0,Y 55.223,Z 519.516,A -85,B 0,C 180,E1 -30572.984,E2 -30572.984} C_VEL
LIN {X 0,Y 64.417,Z 514.512,A -85,B 0,C 180,E1 -30578.031,E2 -30578.031} C_VEL
LIN {X 0,Y 72.973,Z 508.904,A -85,B 0,C 180,E1 -30581.52,E2 -30581.52} C_VEL
LIN {X 0,Y 73.854,Z 507.967,A -85,B 0,C 180,E1 -30583.412,E2 -30583.412} C_VEL
LIN {X 0,Y 74.822,Z 506.496,A -85,B 0,C 180,E1 -30589.172,E2 -30589.172} C_VEL
LIN {X 0,Y 75.716,Z 505.526,A -85,B 0,C 180,E1 -30594.674,E2 -30594.674} C_VEL
LIN {X 0,Y 75.969,Z 505.506,A -85,B 0,C 180,E1 -30600,E2 -30600} C_VEL
LIN {X 0,Y 74.927,Z 506.985,A -85,B 0,C 180,E1 -30605.382,E2 -30605.382} C_VEL
LIN {X 0,Y 74.297,Z 507.987,A -85,B 0,C 180,E1 -30608.344,E2 -30608.344} C_VEL
LIN {X 0,Y 73.243,Z 509.057,A -85,B 0,C 180,E1 -30609.888,E2 -30609.888} C_VEL
LIN {X 0,Y 70.631,Z 511.141,A -85,B 0,C 180,E1 -30611.423,E2 -30611.423} C_VEL
LIN {X 0,Y 67.424,Z 513.28,A -85,B 0,C 180,E1 -30612.238,E2 -30612.238} C_VEL
LIN {X 0,Y 58.43,Z 518.313,A -85,B 0,C 180,E1 -30613.476,E2 -30613.476} C_VEL
LIN {X 0,Y 57.166,Z 518.965,A -85,B 0,C 180,E1 -30613.883,E2 -30613.883} C_VEL
LIN {X 0,Y 48.101,Z 523.378,A -85,B 0,C 180,E1 -30618.244,E2 -30618.244} C_VEL
LIN {X 0,Y 38.782,Z 527.031,A -85,B 0,C 180,E1 -30625.027,E2 -30625.027} C_VEL
LIN {X 0,Y 32.963,Z 528.918,A -85,B 0,C 180,E1 -30631.476,E2 -30631.476} C_VEL
LIN {X 0,Y 23.654,Z 531.388,A -85,B 0,C 180,E1 -30653.539,E2 -30653.539} C_VEL
LIN {X 0,Y 21.024,Z 532.033,A -85,B 0,C 180,E1 -30670.469,E2 -30670.469} C_VEL
LIN {X 0,Y 20.497,Z 532.28,A -85,B 0,C 180,E1 -30689.998,E2 -30689.998} C_VEL
LIN {X 0,Y 21.018,Z 532.014,A -85,B 0,C 180,E1 -30709.533,E2 -30709.533} C_VEL
LIN {X 0,Y 27.812,Z 530.308,A -85,B 0,C 180,E1 -30739.294,E2 -30739.294} C_VEL
LIN {X 0,Y 32.961,Z 528.855,A -85,B 0,C 180,E1 -30748.525,E2 -30748.525} C_VEL
LIN {X 0,Y 41.817,Z 525.851,A -85,B 0,C 180,E1 -30757.57,E2 -30757.57} C_VEL
LIN {X 0,Y 51.298,Z 521.802,A -85,B 0,C 180,E1 -30763.538,E2 -30763.538} C_VEL
LIN {X 0,Y 62.843,Z 515.605,A -85,B 0,C 180,E1 -30768.108,E2 -30768.108} C_VEL
LIN {X 0,Y 66.905,Z 512.994,A -85,B 0,C 180,E1 -30769.695,E2 -30769.695} C_VEL
LIN {X 0,Y 68.661,Z 511.12,A -85,B 0,C 180,E1 -30774.125,E2 -30774.125} C_VEL
LIN {X 0,Y 69.942,Z 509.619,A -85,B 0,C 180,E1 -30780,E2 -30780} C_VEL
LIN {X 0,Y 69.632,Z 509.638,A -85,B 0,C 180,E1 -30785.793,E2 -30785.793} C_VEL
LIN {X 0,Y 68.403,Z 510.692,A -85,B 0,C 180,E1 -30791.858,E2 -30791.858} C_VEL
LIN {X 0,Y 67.565,Z 511.449,A -85,B 0,C 180,E1 -30794.148,E2 -30794.148} C_VEL
LIN {X 0,Y 58.873,Z 516.559,A -85,B 0,C 180,E1 -30797.255,E2 -30797.255} C_VEL
LIN {X 0,Y 49.236,Z 521.217,A -85,B 0,C 180,E1 -30801.904,E2 -30801.904} C_VEL
LIN {X 0,Y 40.067,Z 524.769,A -85,B 0,C 180,E1 -30808.715,E2 -30808.715} C_VEL
LIN {X 0,Y 34.384,Z 526.598,A -85,B 0,C 180,E1 -30815.156,E2 -30815.156} C_VEL
LIN {X 0,Y 25.027,Z 528.935,A -85,B 0,C 180,E1 -30835.833,E2 -30835.833} C_VEL
LIN {X 0,Y 22.088,Z 529.531,A -85,B 0,C 180,E1 -30851.448,E2 -30851.448} C_VEL
LIN {X 0,Y 21.001,Z 529.753,A -85,B 0,C 180,E1 -30870.002,E2 -30870.002} C_VEL
LIN {X 0,Y 22.038,Z 529.556,A -85,B 0,C 180,E1 -30888.599,E2 -30888.599} C_VEL
LIN {X 0,Y 24.984,Z 528.973,A -85,B 0,C 180,E1 -30904.238,E2 -30904.238} C_VEL
LIN {X 0,Y 34.354,Z 526.671,A -85,B 0,C 180,E1 -30924.919,E2 -30924.919} C_VEL
LIN {X 0,Y 43.034,Z 523.82,A -85,B 0,C 180,E1 -30933.927,E2 -30933.927} C_VEL
LIN {X 0,Y 52.388,Z 519.946,A -85,B 0,C 180,E1 -30939.898,E2 -30939.898} C_VEL
LIN {X 0,Y 62.11,Z 514.943,A -85,B 0,C 180,E1 -30944.119,E2 -30944.119} C_VEL
LIN {X 0,Y 67.656,Z 511.58,A -85,B 0,C 180,E1 -30945.976,E2 -30945.976} C_VEL
LIN {X 0,Y 68.52,Z 510.818,A -85,B 0,C 180,E1 -30948.162,E2 -30948.162} C_VEL
LIN {X 0,Y 69.707,Z 509.79,A -85,B 0,C 180,E1 -30954.213,E2 -30954.213} C_VEL
LIN {X 0,Y 69.982,Z 509.802,A -85,B 0,C 180,E1 -30960,E2 -30960} C_VEL
LIN {X 0,Y 68.59,Z 511.408,A -85,B 0,C 180,E1 -30966.226,E2 -30966.226} C_VEL
LIN {X 0,Y 67.011,Z 513.117,A -85,B 0,C 180,E1 -30970.312,E2 -30970.312} C_VEL
LIN {X 0,Y 62.845,Z 515.774,A -85,B 0,C 180,E1 -30971.892,E2 -30971.892} C_VEL
LIN {X 0,Y 57.166,Z 518.965,A -85,B 0,C 180,E1 -30973.883,E2 -30973.883} C_VEL
LIN {X 0,Y 51.942,Z 521.49,A -85,B 0,C 180,E1 -30975.292,E2 -30975.292} C_VEL
LIN {X 0,Y 42.663,Z 524.915,A -85,B 0,C 180,E1 -30976.279,E2 -30976.279} C_VEL
LIN {X 0,Y 33.2,Z 527.651,A -85,B 0,C 180,E1 -30978.057,E2 -30978.057} C_VEL
LIN {X 0,Y 27.812,Z 528.955,A -85,B 0,C 180,E1 -30981.913,E2 -30981.913} C_VEL
LIN {X 0,Y 18.411,Z 530.954,A -85,B 0,C 180,E1 -31000.226,E2 -31000.226} C_VEL
LIN {X 0,Y 14.506,Z 531.6,A -85,B 0,C 180,E1 -31021.018,E2 -31021.018} C_VEL
LIN {X 0,Y 13.392,Z 531.847,A -85,B 0,C 180,E1 -31049.997,E2 -31049.997} C_VEL
LIN {X 0,Y 14.499,Z 531.58,A -85,B 0,C 180,E1 -31078.99,E2 -31078.99} C_VEL
LIN {X 0,Y 23.779,Z 529.873,A -85,B 0,C 180,E1 -31112.454,E2 -31112.454} C_VEL
LIN {X 0,Y 29.862,Z 528.42,A -85,B 0,C 180,E1 -31120.286,E2 -31120.286} C_VEL
LIN {X 0,Y 39.641,Z 525.414,A -85,B 0,C 180,E1 -31127.182,E2 -31127.182} C_VEL
LIN {X 0,Y 52.192,Z 520.207,A -85,B 0,C 180,E1 -31132.262,E2 -31132.262} C_VEL
LIN {X 0,Y 61.952,Z 515.061,A -85,B 0,C 180,E1 -31134.637,E2 -31134.637} C_VEL
LIN {X 0,Y 62.983,Z 514.199,A -85,B 0,C 180,E1 -31137.122,E2 -31137.122} C_VEL
LIN {X 0,Y 63.65,Z 513.578,A -85,B 0,C 180,E1 -31140,E2 -31140} C_VEL
LIN {X 0,Y 63.525,Z 513.447,A -85,B 0,C 180,E1 -31145.315,E2 -31145.315} C_VEL
LIN {X 0,Y 62.335,Z 514.177,A -85,B 0,C 180,E1 -31149.051,E2 -31149.051} C_VEL
LIN {X 0,Y 50.408,Z 520.243,A -85,B 0,C 180,E1 -31152.594,E2 -31152.594} C_VEL
LIN {X 0,Y 40.44,Z 524.152,A -85,B 0,C 180,E1 -31157.093,E2 -31157.093} C_VEL
LIN {X 0,Y 30.854,Z 527.03,A -85,B 0,C 180,E1 -31164.341,E2 -31164.341} C_VEL
LIN {X 0,Y 19.577,Z 529.367,A -85,B 0,C 180,E1 -31184.113,E2 -31184.113} C_VEL
LIN {X 0,Y 15.539,Z 529.963,A -85,B 0,C 180,E1 -31203.112,E2 -31203.112} C_VEL
LIN {X 0,Y 13.913,Z 530.184,A -85,B 0,C 180,E1 -31230.003,E2 -31230.003} C_VEL
LIN {X 0,Y 15.493,Z 529.987,A -85,B 0,C 180,E1 -31256.98,E2 -31256.98} C_VEL
LIN {X 0,Y 19.54,Z 529.404,A -85,B 0,C 180,E1 -31276.003,E2 -31276.003} C_VEL
LIN {X 0,Y 30.828,Z 527.102,A -85,B 0,C 180,E1 -31295.772,E2 -31295.772} C_VEL
LIN {X 0,Y 40.427,Z 524.251,A -85,B 0,C 180,E1 -31302.973,E2 -31302.973} C_VEL
LIN {X 0,Y 50.396,Z 520.376,A -85,B 0,C 180,E1 -31307.475,E2 -31307.475} C_VEL
LIN {X 0,Y 62.407,Z 514.312,A -85,B 0,C 180,E1 -31311.051,E2 -31311.051} C_VEL
LIN {X 0,Y 63.552,Z 513.607,A -85,B 0,C 180,E1 -31314.438,E2 -31314.438} C_VEL
LIN {X 0,Y 63.684,Z 513.734,A -85,B 0,C 180,E1 -31320,E2 -31320} C_VEL
LIN {X 0,Y 62.951,Z 514.423,A -85,B 0,C 180,E1 -31323.196,E2 -31323.196} C_VEL
LIN {X 0,Y 61.923,Z 515.249,A -85,B 0,C 180,E1 -31325.357,E2 -31325.357} C_VEL
LIN {X 0,Y 49.746,Z 521.487,A -85,B 0,C 180,E1 -31328.52,E2 -31328.52} C_VEL
LIN {X 0,Y 39.643,Z 525.505,A -85,B 0,C 180,E1 -31332.818,E2 -31332.818} C_VEL
LIN {X 0,Y 27.812,Z 528.955,A -85,B 0,C 180,E1 -31341.913,E2 -31341.913} C_VEL
LIN {X 0,Y 22.593,Z 530.081,A -85,B 0,C 180,E1 -31347.791,E2 -31347.791} C_VEL
LIN {X 0,Y 17.192,Z 530.834,A -85,B 0,C 180,E1 -31354.638,E2 -31354.638} C_VEL
LIN {X 0,Y 7.513,Z 531.418,A -85,B 0,C 180,E1 -31390.862,E2 -31390.862} C_VEL
LIN {X 0,Y 7.898,Z 531.207,A -85,B 0,C 180,E1 -31453.48,E2 -31453.48} C_VEL
LIN {X 0,Y 14.828,Z 530.485,A -85,B 0,C 180,E1 -31481.425,E2 -31481.425} C_VEL
LIN {X 0,Y 28.265,Z 527.985,A -85,B 0,C 180,E1 -31494.023,E2 -31494.023} C_VEL
LIN {X 0,Y 38.688,Z 524.978,A -85,B 0,C 180,E1 -31497.569,E2 -31497.569} C_VEL
LIN {X 0,Y 50.775,Z 520.21,A -85,B 0,C 180,E1 -31500,E2 -31500} C_VEL
LIN {X 0,Y 56.227,Z 517.587,A -85,B 0,C 180,E1 -31500.665,E2 -31500.665} C_VEL
LIN {X 0,Y 57.332,Z 516.953,A -85,B 0,C 180,E1 -31501.969,E2 -31501.969} C_VEL
LIN {X 0,Y 56.32,Z 517.426,A -85,B 0,C 180,E1 -31503.347,E2 -31503.347} C_VEL
LIN {X 0,Y 45.876,Z 522.081,A -85,B 0,C 180,E1 -31505.276,E2 -31505.276} C_VEL
LIN {X 0,Y 35.507,Z 525.633,A -85,B 0,C 180,E1 -31508.252,E2 -31508.252} C_VEL
LIN {X 0,Y 28.668,Z 527.462,A -85,B 0,C 180,E1 -31511.312,E2 -31511.312} C_VEL
LIN {X 0,Y 15.505,Z 529.798,A -85,B 0,C 180,E1 -31524.97,E2 -31524.97} C_VEL
LIN {X 0,Y 9.764,Z 530.394,A -85,B 0,C 180,E1 -31543.969,E2 -31543.969} C_VEL
LIN {X 0,Y 6.833,Z 530.615,A -85,B 0,C 180,E1 -31590.006,E2 -31590.006} C_VEL
LIN {X 0,Y 9.723,Z 530.418,A -85,B 0,C 180,E1 -31636.295,E2 -31636.295} C_VEL
LIN {X 0,Y 15.478,Z 529.836,A -85,B 0,C 180,E1 -31655.258,E2 -31655.258} C_VEL
LIN {X 0,Y 28.659,Z 527.533,A -85,B 0,C 180,E1 -31668.796,E2 -31668.796} C_VEL
LIN {X 0,Y 38.945,Z 524.682,A -85,B 0,C 180,E1 -31673,E2 -31673} C_VEL
LIN {X 0,Y 49.348,Z 520.805,A -85,B 0,C 180,E1 -31675.518,E2 -31675.518} C_VEL
LIN {X 0,Y 56.313,Z 517.593,A -85,B 0,C 180,E1 -31676.795,E2 -31676.795} C_VEL
LIN {X 0,Y 57.357,Z 517.114,A -85,B 0,C 180,E1 -31678.347,E2 -31678.347} C_VEL
LIN {X 0,Y 56.229,Z 517.745,A -85,B 0,C 180,E1 -31679.334,E2 -31679.334} C_VEL
LIN {X 0,Y 45.689,Z 522.507,A -85,B 0,C 180,E1 -31680.915,E2 -31680.915} C_VEL
LIN {X 0,Y 35.206,Z 526.163,A -85,B 0,C 180,E1 -31683.479,E2 -31683.479} C_VEL
LIN {X 0,Y 25.082,Z 528.714,A -85,B 0,C 180,E1 -31687.703,E2 -31687.703} C_VEL
LIN {X 0,Y 14.838,Z 530.519,A -85,B 0,C 180,E1 -31698.67,E2 -31698.67} C_VEL
LIN {X 0,Y 8.974,Z 531.167,A -85,B 0,C 180,E1 -31718.439,E2 -31718.439} C_VEL
LIN {X 0,Y 6.279,Z 531.414,A -85,B 0,C 180,E1 -31769.993,E2 -31769.993} C_VEL
LIN {X 0,Y 7.898,Z 531.207,A -85,B 0,C 180,E1 -31813.48,E2 -31813.48} C_VEL
LIN {X 0,Y 9.314,Z 533.206,A -85,B 0,C 180,E1 -31823.633,E2 -31823.633} C_VEL
LIN {X 0,Y 9.314,Z 600,A -85,B 0,C 180,E1 -31823.633,E2 -31823.633} C_VEL
LIN {X 0,Y 9.314,Z 600,A -85,B 0,C 180,E1 -31823.633,E2 -31823.633}

QRS_NEXT_CUT()

QRS_NEXT()
QRS_HOME()

END
